Universal Robots PolyScope program: Safe_Home_BeforeStart.urp

Program Safe_Home_BeforeStart (installation=default directory=/programs createdIn=3.2.18744.0 lastSavedIn=5.9.1.1031110 robotSerialNumber=20195501059)
Calibrated DH parameters: a=[0.000146, -0.418764, -0.053981, 0.000058, -0.000023, 0]; d=[0.162545, 37.319448, -206.067439, 168.881546, 0.09955, 0.099464]; alpha=[1.57004, -0.001979, 0.002304, 1.570607, -1.57066, 0]; deltaTheta=[0, -0.174616, -1.258233, 1.432844, -0.000001, 0]
BeforeStart
  Folder Safe Home Folder
    'Read robot current position'
    start_pose := get_actual_tcp_pose()
    MoveL speed 250 mm/s, acceleration 1200 mm/s^2 (useActiveTCP=true) feature=Base
      'First pose is current pose'
      'Variable position'
      Waypoint Waypoint (Variable): variable=start_pose
    'Break start pose into directions'
    start_x := start_pose[0]
    start_y := start_pose[1]
    start_z := start_pose[2]
    'If TCP is inside box'
    If (start_x≥0.2) and (start_y≥0.1)
      'Move to safe pos. 50 mm above box edge'
      Safe_Z_value := 0.350
      'Same as start pose, but with altered Z-value'
      Safe_Pose := p[start_pose[0],start_pose[1],Safe_Z_value,start_pose[3],start_pose[4],start_pose[5]]
      MoveL speed 250 mm/s, acceleration 1200 mm/s^2 (useActiveTCP=true) feature=Base
        Waypoint Waypoint (Variable): variable=Safe_Pose
Robot Program (runOnlyOnce=false)
  MoveJ speed 60 deg/s, acceleration 80 deg/s^2 (useActiveTCP=false) feature=Base
    Waypoint Normal_start: TCP in base x=116.908 y=-391.817 z=399.559 mm, rx=2.4514 ry=1.3085 rz=-0.4986 rad; joints [89.773, -105.294, 124.331, -134.949, 261.315, 121.598] deg
